FUNCTION A_INT : ST_Arg
VAR_INPUT
	nNumber	: REFERENCE TO INT;
END_VAR

IF __ISVALIDREF(nNumber) THEN
	A_INT.eType := E_ArgType.IntArg;
	A_INT.pData := ADR(nNumber);
	A_INT.nSize := SIZEOF(INT);
END_IF

END_FUNCTION

(* stored: Version 1.1.0.1, ProductVersion 3.1.4024.15
   POU A_INT: Id {d3c2d0e4-a1a1-4b34-933b-f53443c0192e}, SpecialFunc None *)
